// TIA Portal V20 export
DATA_BLOCK "GLOBAL_Sensing_HMI_IF_DB"   // DB217
{ S7_Optimized_Access := 'TRUE' }
// stored: AutoNumber false, MemoryReserve 100
   VAR
      Sensing { S7_SetPoint := 'True'} : Array[0..1] of "KEYENCE_HMI_IF_UDT";
   END_VAR
BEGIN
END_DATA_BLOCK
